// TIA Portal V19 export
FUNCTION "LAF_MapUnitStatusToSequence" : Void   // FC70, LAD
TITLE = LAF_MapUnitStatusToSequence
AUTHOR : Siemens Digital Industries
FAMILY : LAF
VERSION : 1.2
// Connect the unit status signals to the sequencer interface.
// stored: Access Published, IsIECCheckEnabled true, SetENOAutomatically false
   VAR_INPUT
      interruptJobInStopping : Bool;   // Configuration if the current job should be interrupted when the unit status changes to stopping. New jobs could be executed afterwards.
      interruptJobInHolding : Bool;   // Configuration if the current job should be interrupted when the unit status changes to holding. New jobs could be executed afterwards.
      interruptJobInSuspending : Bool;   // Configuration if the current job should be interrupted when the unit status changes to suspending. New jobs could be executed afterwards.
      interruptJobInCompleting : Bool;   // Configuration if the current job should be interrupted when the unit status changes to completing. New jobs could be executed afterwards.
      unitStatus : "LAF_typeUnitStatus";
   END_VAR
   VAR_IN_OUT
      jobs : "LAF_typeJobs";
      sequence : "LAF_typeSequence";
   END_VAR
BEGIN

REGION Network 1: BLOCK INFO HEADER
   // SIEMENS AG / (c)Copyright 2024
   // ------------------------------------------------------------------------------
   // Title:            LAF_MapUnitStatusToSequence
   // Comment/Function: Connect the unit status signals to the sequencer interface.
   // Library/Family:   Library of Automation Framework
   // Author:                Siemens Digital Industry
   // Tested with:       S7-PLCSIM Advanced 6.0
   // Engineering:      TIA Portal V19
   // Restrictions:       ---
   // Requirements:   ---
   // ------------------------------------------------------------------------------
   // Change log table:
   // Version  | Date       | Expert in charge       | Changes applied
   // ---------|------------|------------------------|------------------------------
   // 01.01.00 | 21.06.2024 | SIMATIC Systems Support | First released version
   // 01.02.00 | 30.09.2024 | SIMATIC Systems Support | Block information properties updated and optimized code
END_REGION

REGION Network 2: DESCRIPTION
   // The LAF_MapUnitStatusToSequence function block is used to connect the unit status signals to the sequencer interface. If the active Unit Mode is Manual, the HMI interface signals are used to control the sequence.
   // The block should be adapted if another Unit Control Manager is used.
END_REGION

REGION Network 3: Select Sequence Mode Production
   // Set the Sequencer in Automatic Mode.
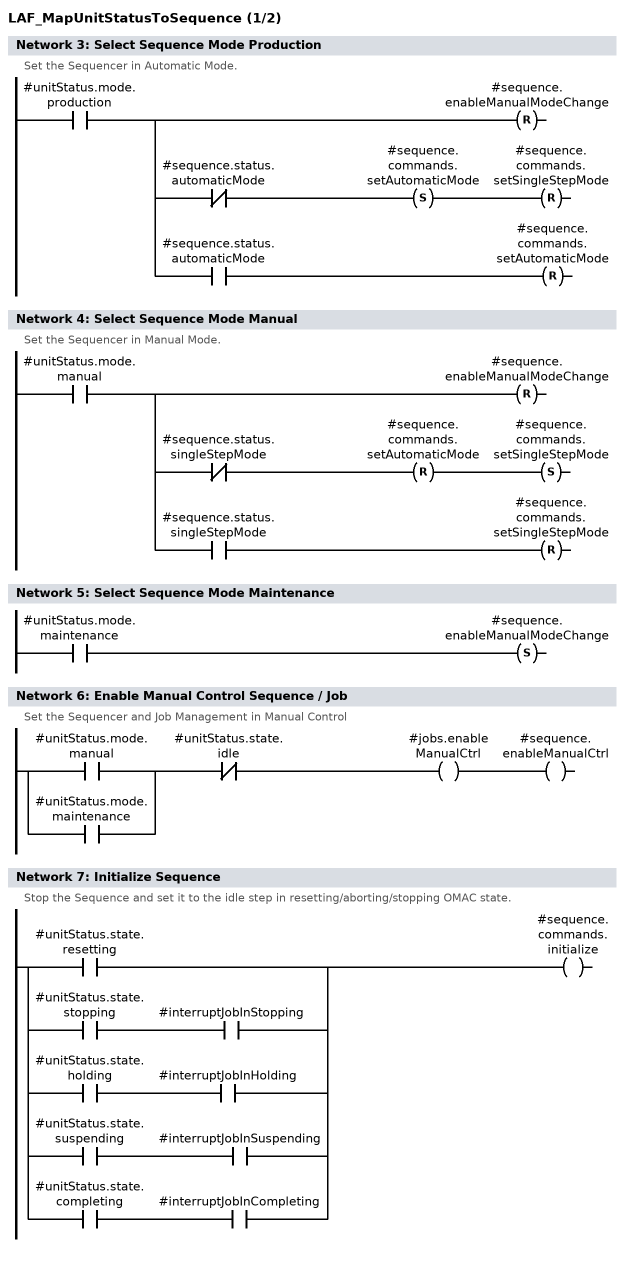
   RUNG wire#powerrail
      Contact( #unitStatus.mode.production )
      wire#w1
      R_Coil( #sequence.enableManualModeChange )
   END_RUNG
   RUNG wire#w1
      I_Contact( #sequence.status.automaticMode )
      S_Coil( #sequence.commands.setAutomaticMode )
      R_Coil( #sequence.commands.setSingleStepMode )
   END_RUNG
   RUNG wire#w1
      Contact( #sequence.status.automaticMode )
      R_Coil( #sequence.commands.setAutomaticMode )
   END_RUNG
   // the same network as SCL:
   IF #unitStatus.mode.production THEN #sequence.enableManualModeChange := FALSE; END_IF;
   IF #unitStatus.mode.production AND NOT #sequence.status.automaticMode THEN
       #sequence.commands.setAutomaticMode := TRUE;
       #sequence.commands.setSingleStepMode := FALSE;
   END_IF;
   IF #unitStatus.mode.production AND #sequence.status.automaticMode THEN
       #sequence.commands.setAutomaticMode := FALSE;
   END_IF;
END_REGION

REGION Network 4: Select Sequence Mode Manual
   // Set the Sequencer in Manual Mode.
   RUNG wire#powerrail
      Contact( #unitStatus.mode.manual )
      wire#w1
      R_Coil( #sequence.enableManualModeChange )
   END_RUNG
   RUNG wire#w1
      I_Contact( #sequence.status.singleStepMode )
      R_Coil( #sequence.commands.setAutomaticMode )
      S_Coil( #sequence.commands.setSingleStepMode )
   END_RUNG
   RUNG wire#w1
      Contact( #sequence.status.singleStepMode )
      R_Coil( #sequence.commands.setSingleStepMode )
   END_RUNG
   // the same network as SCL:
   IF #unitStatus.mode.manual THEN #sequence.enableManualModeChange := FALSE; END_IF;
   IF #unitStatus.mode.manual AND NOT #sequence.status.singleStepMode THEN
       #sequence.commands.setAutomaticMode := FALSE;
       #sequence.commands.setSingleStepMode := TRUE;
   END_IF;
   IF #unitStatus.mode.manual AND #sequence.status.singleStepMode THEN
       #sequence.commands.setSingleStepMode := FALSE;
   END_IF;
END_REGION

REGION Network 5: Select Sequence Mode Maintenance
   RUNG wire#powerrail
      Contact( #unitStatus.mode.maintenance )
      S_Coil( #sequence.enableManualModeChange )
   END_RUNG
   // the same network as SCL:
   IF #unitStatus.mode.maintenance THEN #sequence.enableManualModeChange := TRUE; END_IF;
END_REGION

REGION Network 6: Enable Manual Control Sequence / Job
   // Set the Sequencer and Job Management in Manual Control
   RUNG wire#powerrail
      Contact( #unitStatus.mode.manual )
      wire#w1
      I_Contact( #unitStatus.state.idle )
      Coil( #jobs.enableManualCtrl )
      Coil( #sequence.enableManualCtrl )
   END_RUNG
   RUNG wire#powerrail
      Contact( #unitStatus.mode.maintenance )
   END_RUNG wire#w1
   // the same network as SCL:
   #jobs.enableManualCtrl := (#unitStatus.mode.manual OR #unitStatus.mode.maintenance) AND NOT #unitStatus.state.idle;
   #sequence.enableManualCtrl := #jobs.enableManualCtrl;
END_REGION

REGION Network 7: Initialize Sequence
   // Stop the Sequence and set it to the idle step in resetting/aborting/stopping OMAC state.
   RUNG wire#powerrail
      Contact( #unitStatus.state.resetting )
      wire#w1
      Coil( #sequence.commands.initialize )
   END_RUNG
   RUNG wire#powerrail
      Contact( #unitStatus.state.stopping )
      Contact( #interruptJobInStopping )
   END_RUNG wire#w1
   RUNG wire#powerrail
      Contact( #unitStatus.state.holding )
      Contact( #interruptJobInHolding )
   END_RUNG wire#w1
   RUNG wire#powerrail
      Contact( #unitStatus.state.suspending )
      Contact( #interruptJobInSuspending )
   END_RUNG wire#w1
   RUNG wire#powerrail
      Contact( #unitStatus.state.completing )
      Contact( #interruptJobInCompleting )
   END_RUNG wire#w1
   // the same network as SCL:
   #sequence.commands.initialize := #unitStatus.state.resetting OR (#unitStatus.state.stopping AND #interruptJobInStopping) OR (#unitStatus.state.holding AND #interruptJobInHolding) OR (#unitStatus.state.suspending AND #interruptJobInSuspending) OR (#unitStatus.state.completing AND #interruptJobInCompleting);
END_REGION

REGION Network 8: Immediately Stop the Sequence
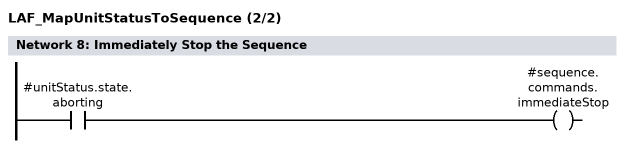
   RUNG wire#powerrail
      Contact( #unitStatus.state.aborting )
      Coil( #sequence.commands.immediateStop )
   END_RUNG
   // the same network as SCL:
   #sequence.commands.immediateStop := #unitStatus.state.aborting;
END_REGION
END_FUNCTION
